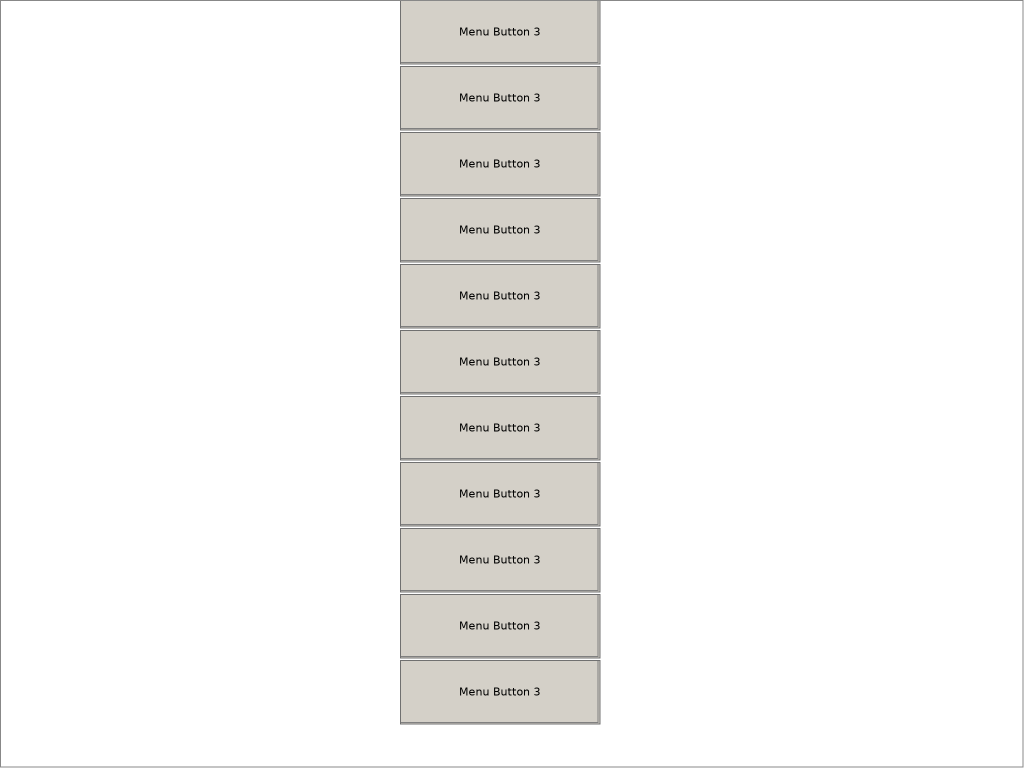
VISUALIZATION PopupMenu3  // 1024x768
    Button (400,0 200x64), "Menu Button 3"
        OnMouseClick: CloseDialog Dialog=PopupMenu3, Result=None, NumpadKeypadSet=True
    Button (400,66 200x64), "Menu Button 3"
        OnMouseClick: CloseDialog Dialog=PopupMenu3, Result=None, NumpadKeypadSet=True
    Button (400,132 200x64), "Menu Button 3"
        OnMouseClick: CloseDialog Dialog=PopupMenu3, Result=None, NumpadKeypadSet=True
    Button (400,198 200x64), "Menu Button 3"
        OnMouseClick: CloseDialog Dialog=PopupMenu3, Result=None, NumpadKeypadSet=True
    Button (400,264 200x64), "Menu Button 3"
        OnMouseClick: CloseDialog Dialog=PopupMenu3, Result=None, NumpadKeypadSet=True
    Button (400,330 200x64), "Menu Button 3"
        OnMouseClick: CloseDialog Dialog=PopupMenu3, Result=None, NumpadKeypadSet=True
    Button (400,396 200x64), "Menu Button 3"
        OnMouseClick: CloseDialog Dialog=PopupMenu3, Result=None, NumpadKeypadSet=True
    Button (400,462 200x64), "Menu Button 3"
        OnMouseClick: CloseDialog Dialog=PopupMenu3, Result=None, NumpadKeypadSet=True
    Button (400,528 200x64), "Menu Button 3"
        OnMouseClick: CloseDialog Dialog=PopupMenu3, Result=None, NumpadKeypadSet=True
    Button (400,594 200x64), "Menu Button 3"
        OnMouseClick: CloseDialog Dialog=PopupMenu3, Result=None, NumpadKeypadSet=True
    Button (400,660 200x64), "Menu Button 3"
        OnMouseClick: CloseDialog Dialog=PopupMenu3, Result=None, NumpadKeypadSet=True
    InvisibleInput (600,0 425x768)
        OnMouseClick: CloseDialog Dialog=PopupMenu3, Result=OK, NumpadKeypadSet=True
    InvisibleInput (0,0 400x768)
        OnMouseClick: CloseDialog Dialog=PopupMenu3, Result=OK, NumpadKeypadSet=True
    InvisibleInput (400,725 203x44)
        OnMouseClick: CloseDialog Dialog=PopupMenu3, Result=OK, NumpadKeypadSet=True
END_VISUALIZATION

(* stored: Version 1.1.0.1, ProductVersion 3.1.4024.11
   Visu PopupMenu3: Id {f77d2e83-0b36-0d53-07a2-e8866b15d9de} *)
